Staubli VAL3: RefreshBelt.pgx

program RefreshBelt()
begin
  //
  gotoxy(20,1)
  put("--砂带信息--")
  gotoxy(20,3)
  put("补偿量:"+toString(".3",PublicData:nSumCompen)+"  ")
  gotoxy(20,4)
  put("补偿次数:"+toString("4",PublicData:nCompenCount)+"  ")
end
